{attribute addProperty BoxType "EL2521-0000-1019"}
{attribute addProperty Id "StatusAT %I*Status_4EB9B0BC1620Counter_valueAT %I*UINT16217"}
{attribute addProperty CRC "4039838391"}
{attribute addProperty SizeInBites "32"}
{attribute addProperty SizeInBytes "4"}
TYPE ENC_Status_compact_F0CB0AB7 :
STRUCT
	{attribute addProperty Name "Status"}
	Status AT %I* : Status_4EB9B0BC;
	{attribute addProperty Name "Counter_value"}
	Counter_value AT %I* : UINT;
END_STRUCT
END_TYPE

(* stored: Version 1.2.0.0, ProductVersion 3.1.4024.9
   DUT ENC_Status_compact_F0CB0AB7: Id {2736bb3c-de2e-410c-8fe5-9da75d9dbebe} *)
